# EPICS autosave request: dxp/trunk/iocBoot/iocXMAP/auto_settings12.req
file "dxpSystem_settings.req"           P=$(P)
file "dxpMED_settings.req"              P=$(P)
file "dxpXMAP_settings.req",            P=$(P)
file "dxpHighLevel_settings.req",       P=$(P), R=dxp1:
file "dxpHighLevel_settings.req",       P=$(P), R=dxp2:
file "dxpHighLevel_settings.req",       P=$(P), R=dxp3:
file "dxpHighLevel_settings.req",       P=$(P), R=dxp4:
file "dxpHighLevel_settings.req",       P=$(P), R=dxp5:
file "dxpHighLevel_settings.req",       P=$(P), R=dxp6:
file "dxpHighLevel_settings.req",       P=$(P), R=dxp7:
file "dxpHighLevel_settings.req",       P=$(P), R=dxp8:
file "dxpHighLevel_settings.req",       P=$(P), R=dxp9:
file "dxpHighLevel_settings.req",       P=$(P), R=dxp10:
file "dxpHighLevel_settings.req",       P=$(P), R=dxp11:
file "dxpHighLevel_settings.req",       P=$(P), R=dxp12:
file "dxpSCA_16_settings.req",          P=$(P), R=dxp1:
file "dxpSCA_16_settings.req",          P=$(P), R=dxp2:
file "dxpSCA_16_settings.req",          P=$(P), R=dxp3:
file "dxpSCA_16_settings.req",          P=$(P), R=dxp4:
file "dxpSCA_16_settings.req",          P=$(P), R=dxp5:
file "dxpSCA_16_settings.req",          P=$(P), R=dxp6:
file "dxpSCA_16_settings.req",          P=$(P), R=dxp7:
file "dxpSCA_16_settings.req",          P=$(P), R=dxp8:
file "dxpSCA_16_settings.req",          P=$(P), R=dxp9:
file "dxpSCA_16_settings.req",          P=$(P), R=dxp10:
file "dxpSCA_16_settings.req",          P=$(P), R=dxp11:
file "dxpSCA_16_settings.req",          P=$(P), R=dxp12:
file "simple_mca_settings.req",         P=$(P), M=mca1
file "simple_mca_settings.req",         P=$(P), M=mca2
file "simple_mca_settings.req",         P=$(P), M=mca3
file "simple_mca_settings.req",         P=$(P), M=mca4
file "simple_mca_settings.req",         P=$(P), M=mca5
file "simple_mca_settings.req",         P=$(P), M=mca6
file "simple_mca_settings.req",         P=$(P), M=mca7
file "simple_mca_settings.req",         P=$(P), M=mca8
file "simple_mca_settings.req",         P=$(P), M=mca9
file "simple_mca_settings.req",         P=$(P), M=mca10
file "simple_mca_settings.req",         P=$(P), M=mca11
file "simple_mca_settings.req",         P=$(P), M=mca12

file "NDPluginBase_settings.req",       P=$(P), R=netCDF1:
file "NDFile_settings.req",             P=$(P), R=netCDF1:

file scan_settings.req                  P=$(P), S=scan1
file scan_settings.req                  P=$(P), S=scan2
file scan_settings.req                  P=$(P), S=scan3
file scan_settings.req                  P=$(P), S=scan4
file scan_settings.req                  P=$(P), S=scanH

file saveData_settings.req              P=$(P)
